// TIA Portal V18 export
FUNCTION_BLOCK "FB0-MR_Quantity Control_1"   // FB13, LAD
{ S7_Optimized_Access := 'TRUE' }
VERSION : 0.1
// stored: AutoNumber false, IsIECCheckEnabled false, IsRetainMemResEnabled false, MemoryReserve 100, SetENOAutomatically false, UDAEnableTagReadback false
   VAR_INPUT
      RatioCheckMode : Int;
      AcceptValue : Bool;
      "Mixing Ratio 100:B" : Real;
      "Qty A set" : Real;
      "Qty B set" : Real;
      "Pump size A" : Real;
      "Pump size B" : Real;
      RatioCheckStarted : Bool;
      DeleteCalibrationA : Bool;
      DeleteCalibrationB : Bool;
   END_VAR
   VAR_OUTPUT
      "Max. Mixed quantity" : Real;
      "Pump Capacity A cc/rev" : Real;
      "Pump capacity B cc/rev" : Real;
      "cc/rev A" : Real;
      "cc/rev B" : Real;
      "pump adj. ratio A" : Real;
      "pump adj. ratio B" : Real;
      "Total Deviation A" : Real;
      "Total Deviation B" : Real;
      "Current Deviation A" : Real;
      "Current Deviation B" : Real;
      AllowedMaxAQtyOn2kMetering : Real;
      AllowedMaxBQtyOn2kMetering_1 : Real;
   END_VAR
   VAR_IN_OUT
      "Qty real A" : Real;
      "Qty real B" : Real;
   END_VAR
   VAR RETAIN
      "Last_Cc/rev_A" : Real;
      "Last_Cc/rev_B" : Real;
   END_VAR
   VAR
      "A_Qty/rev_Theor" : Real;
      "B_Qty/rev_Theor" : Real;
      A_Calc_Ref_rev : Real;
      B_Calc_Ref_rev : Real;
      A_Total_Deviation : Real;
      B_Total_Deviation : Real;
   END_VAR
   VAR RETAIN
      B_Current_Deviation : Real;
      A_Current_Deviation : Real;
      "CC/rev actual A" : Real;
      "CC/rev actual B" : Real;
   END_VAR
   VAR
      "A_cc/revStatic_Found" : Real;
      "B_cc/revStatic_Found" : Real;
      "cc/rev calc A" : Real;
      "cc/rev calc B" : Real;
      "Maximum capacity Pump A" : Real;
      "Maximum capacity Pump B" : Real;
      "Individual quantity A MR" : Real;
      "Individual quantity B1 MR" : Real;
      "Individual quantity B MR" : Real;
      "capacity difference" : Real;
      "Ratio margin" : Real;
      "Ratio/100" : Real;
      "Pump cc/rev A" : Real;
      "pump cc/rev B" : Real;
      "A Quantity Compensated" : Real;
      "Quantity A Per ratio" : Real;
      Temp_1 : Bool;
      Last_DeviationA : Real;
      Last_DeviationB : Real;
   END_VAR
   VAR_TEMP   // added for the SCL form of the ladder/FBD networks
      _w1 : Bool;
   END_VAR
BEGIN

REGION Network 1
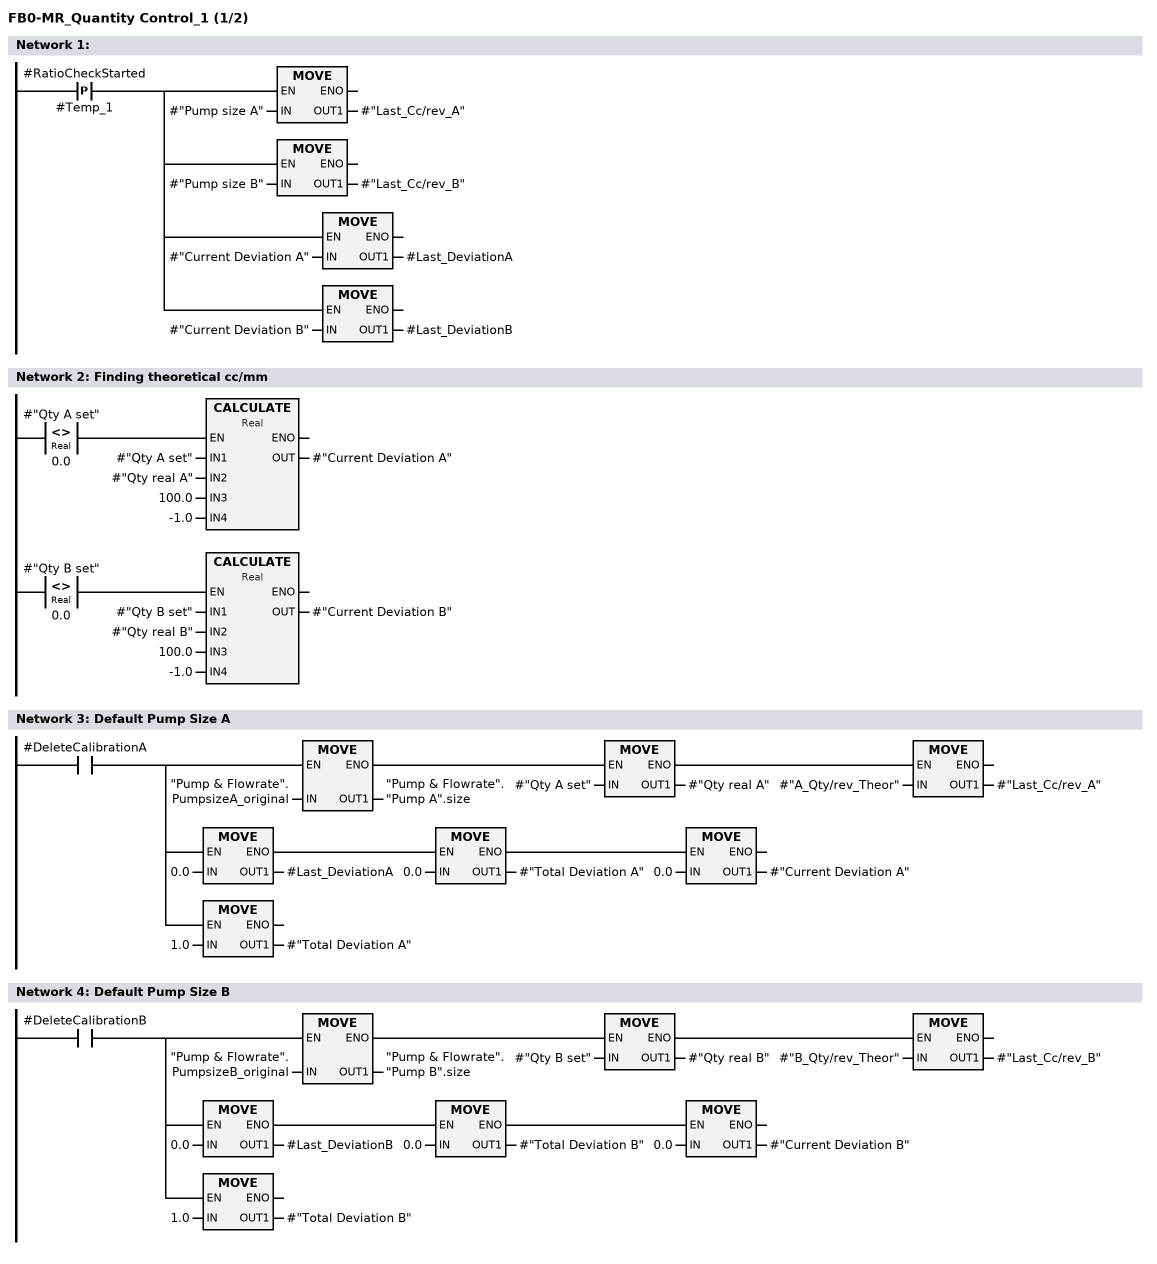
   RUNG wire#powerrail
      P_Contact(operand := #RatioCheckStarted, bit := #Temp_1)
      wire#w1
      Move(in := #"Pump size A", out1 => #"Last_Cc/rev_A")
   END_RUNG
   RUNG wire#w1
      Move(in := #"Pump size B", out1 => #"Last_Cc/rev_B")
   END_RUNG
   RUNG wire#w1
      Move(in := #"Current Deviation A", out1 => #Last_DeviationA)
   END_RUNG
   RUNG wire#w1
      Move(in := #"Current Deviation B", out1 => #Last_DeviationB)
   END_RUNG
   // the same network as SCL:
   #_w1 := #RatioCheckStarted AND NOT #Temp_1;   // rising edge of #RatioCheckStarted
   #Temp_1 := #RatioCheckStarted;
   IF #_w1 THEN
       #"Last_Cc/rev_A" := #"Pump size A";
       #"Last_Cc/rev_B" := #"Pump size B";
       #Last_DeviationA := #"Current Deviation A";
       #Last_DeviationB := #"Current Deviation B";
   END_IF;
END_REGION

REGION Network 2: Finding theoretical cc/mm
   RUNG wire#powerrail
      { S7_Templates := "SrcType := Real" } NE_Contact(in1 := #"Qty A set", in2 := 0.0)
      { S7_Templates := "SrcType := Real"; S7_Expression := "((IN1-IN2)/(IN1/IN3))*(IN4)" } Calculate(in1 := #"Qty A set", in2 := #"Qty real A", in3 := 100.0, in4 := -1.0, out => #"Current Deviation A")
   END_RUNG
   RUNG wire#powerrail
      { S7_Templates := "SrcType := Real" } NE_Contact(in1 := #"Qty B set", in2 := 0.0)
      { S7_Templates := "SrcType := Real"; S7_Expression := "(IN1-IN2)/(IN1/IN3)*(IN4)" } Calculate(in1 := #"Qty B set", in2 := #"Qty real B", in3 := 100.0, in4 := -1.0, out => #"Current Deviation B")
   END_RUNG
   // the same network as SCL:
   IF #"Qty A set" <> 0.0 THEN
       #"Current Deviation A" := ((#"Qty A set"-#"Qty real A")/(#"Qty A set"/100.0))*((-1.0));
   END_IF;
   IF #"Qty B set" <> 0.0 THEN
       #"Current Deviation B" := (#"Qty B set"-#"Qty real B")/(#"Qty B set"/100.0)*((-1.0));
   END_IF;
END_REGION

REGION Network 3: Default Pump Size A
   IF #DeleteCalibrationA THEN
       "Pump & Flowrate"."Pump A".size := "Pump & Flowrate".PumpsizeA_original;
       #"Qty real A" := #"Qty A set";
       #"Last_Cc/rev_A" := #"A_Qty/rev_Theor";
       #Last_DeviationA := 0.0;
       #"Total Deviation A" := 0.0;
       #"Current Deviation A" := 0.0;
       #"Total Deviation A" := 1.0;
   END_IF;
END_REGION

REGION Network 4: Default Pump Size B
   IF #DeleteCalibrationB THEN
       "Pump & Flowrate"."Pump B".size := "Pump & Flowrate".PumpsizeB_original;
       #"Qty real B" := #"Qty B set";
       #"Last_Cc/rev_B" := #"B_Qty/rev_Theor";
       #Last_DeviationB := 0.0;
       #"Total Deviation B" := 0.0;
       #"Current Deviation B" := 0.0;
       #"Total Deviation B" := 1.0;
   END_IF;
END_REGION

REGION Network 5
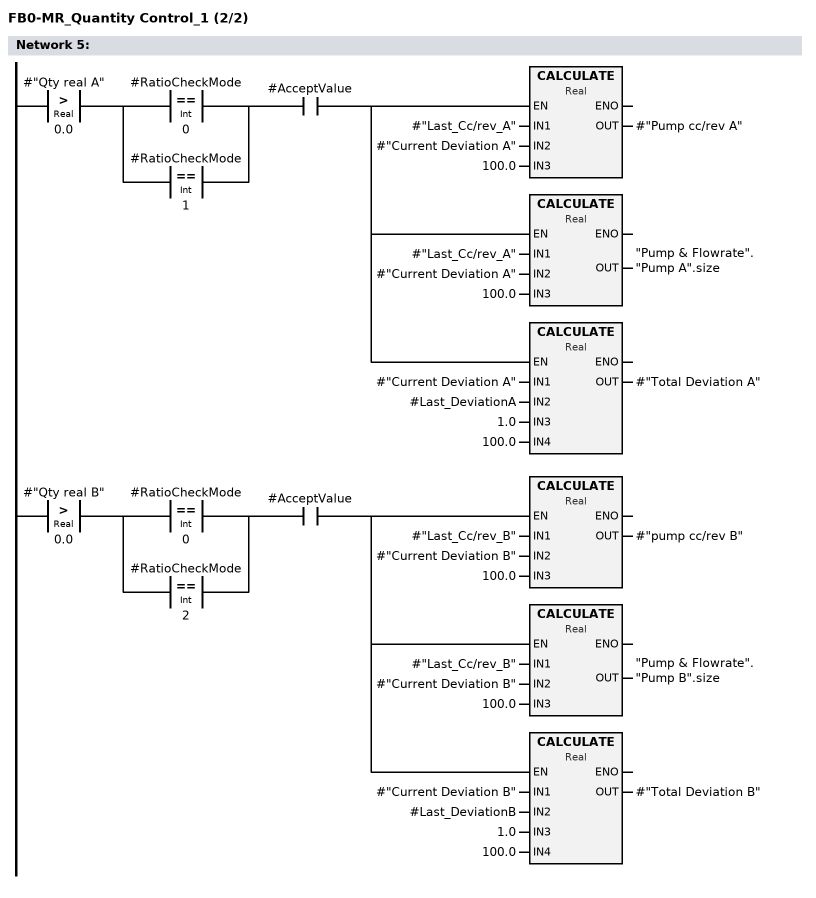
   IF (#"Qty real A" > 0.0) AND ((#RatioCheckMode = 0) OR (#RatioCheckMode = 1)) AND #AcceptValue THEN
       #"Pump cc/rev A" := #"Last_Cc/rev_A"+(#"Last_Cc/rev_A"*(#"Current Deviation A"/100.0));
       "Pump & Flowrate"."Pump A".size := #"Last_Cc/rev_A"+(#"Last_Cc/rev_A"*(#"Current Deviation A"/100.0));
       #"Total Deviation A" := 1.0-((#"Current Deviation A"+#Last_DeviationA)/100.0);
   END_IF;
   IF (#"Qty real B" > 0.0) AND ((#RatioCheckMode = 0) OR (#RatioCheckMode = 2)) AND #AcceptValue THEN
       #"pump cc/rev B" := #"Last_Cc/rev_B"+(#"Last_Cc/rev_B"*(#"Current Deviation B"/100.0));
       "Pump & Flowrate"."Pump B".size := #"Last_Cc/rev_B"+(#"Last_Cc/rev_B"*(#"Current Deviation B"/100.0));
       #"Total Deviation B" := 1.0-((#"Current Deviation B"+#Last_DeviationB)/100.0);
   END_IF;
END_REGION
END_FUNCTION_BLOCK
